// TIA Portal V20 export
DATA_BLOCK "LBP_InternalDB8"   // DB8
TITLE = Internal DB for basic program / DB interne pour programme de base
{ S7_Optimized_Access := 'FALSE' }
AUTHOR : SINUMERIK
FAMILY : SINUMERIK_ONE
VERSION : 6.24
// DB only for internal use in the basic program / DB réservé à l'utilisation interne dans le programme de base
// stored: AutoNumber false
   VAR RETAIN
      DoNotUse0 : DWord;
      Reserved4 : Array[4..7] of Byte;
      FirstCycle : Byte;   // not used / non utilisé
      InternalUse9_0 : Bool;
      InternalUse9_1 : Bool;
      AL_404031 : Bool;
      InternalUse9_3 : Bool;
      InternalUse10 : Array[1..10] of Bool;
      InternalUse12 : SInt;
      InternalUse14 : Array[1..10] of Bool;
      InternalUse16 : SInt;
      InternalUse18 : Array[1..10] of Bool;
      InternalUse20 : Array[1..10] of Bool;
      Reserved22 : Array[22..53] of Byte;   // not used / non utilisé
      InternalUse54 : DWord;
      InternalUse58 : DWord;
      DoNotUse62 : DWord;
      Reserved66 : Array[66..75] of Byte;
      InternalUse76 : DWord;
      InternalUse80 : DInt;   // internal use only / réservé à l'utilisation interne
      InternalUse84 : LReal;   // internal use only / réservé à l'utilisation interne
      MinCycleTime : Int;   // not used / non utilisé
      AdaptTime : Int;   // not used / non utilisé
      ActCycleTime : Int;   // not used / non utilisé
      InternalUse98 : HW_ANY;   // internal use only / réservé à l'utilisation interne
      InternalUse100 : LReal;
   END_VAR
BEGIN
END_DATA_BLOCK
